PROGRAM Main
VAR
	testSlave : TestTwin(ipAddress := '127.0.0.1', tcpPort := 503, unitId := 255);
END_VAR

testSlave.CyclicCall();

END_PROGRAM

(* stored: Version 1.1.0.1, ProductVersion 3.1.4024.12
   POU Main: Id {f82a1f00-d9e1-4635-8047-480831a8854c}, SpecialFunc None *)
